FUNCTION_BLOCK SKILL_Gate (* Command authority for one skill: procedure calls only while the unit runs; OPC UA commands only from the occupation owner outside Production; unit control always *)
  (* Standard: 61499-2 *)
  (* Version 2.0, 2026-09-27, Project contributors, Filling cell reference model *)
  PACKAGE fillingcell;
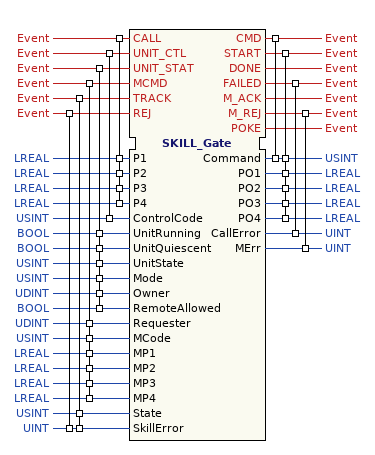
  EVENT_INPUT
    CALL WITH P1, P2, P3, P4;
    UNIT_CTL WITH ControlCode;
    UNIT_STAT WITH UnitRunning, UnitQuiescent, UnitState, Mode, Owner, RemoteAllowed;
    MCMD WITH Requester, MCode, MP1, MP2, MP3, MP4;
    TRACK WITH State, SkillError;
    REJ WITH SkillError;
  END_EVENT
  EVENT_OUTPUT
    CMD WITH Command;
    START WITH Command, PO1, PO2, PO3, PO4;
    DONE;
    FAILED WITH CallError;
    M_ACK;
    M_REJ WITH MErr;
    POKE;
  END_EVENT
  VAR_INPUT
    P1 : LREAL;
    P2 : LREAL;
    P3 : LREAL;
    P4 : LREAL;
    ControlCode : USINT;
    UnitRunning : BOOL;
    UnitQuiescent : BOOL;
    UnitState : USINT;
    Mode : USINT;
    Owner : UDINT;
    RemoteAllowed : BOOL;
    Requester : UDINT;
    MCode : USINT;
    MP1 : LREAL;
    MP2 : LREAL;
    MP3 : LREAL;
    MP4 : LREAL;
    State : USINT := 4;
    SkillError : UINT;
  END_VAR
  VAR_OUTPUT
    Command : USINT;
    PO1 : LREAL;
    PO2 : LREAL;
    PO3 : LREAL;
    PO4 : LREAL;
    CallError : UINT;
    MErr : UINT;
  END_VAR
  VAR
    CallPending : BOOL;
    PendingStart : BOOL;
    MPending : BOOL;
    ManualOK : BOOL;
    Valid : BOOL;
  END_VAR
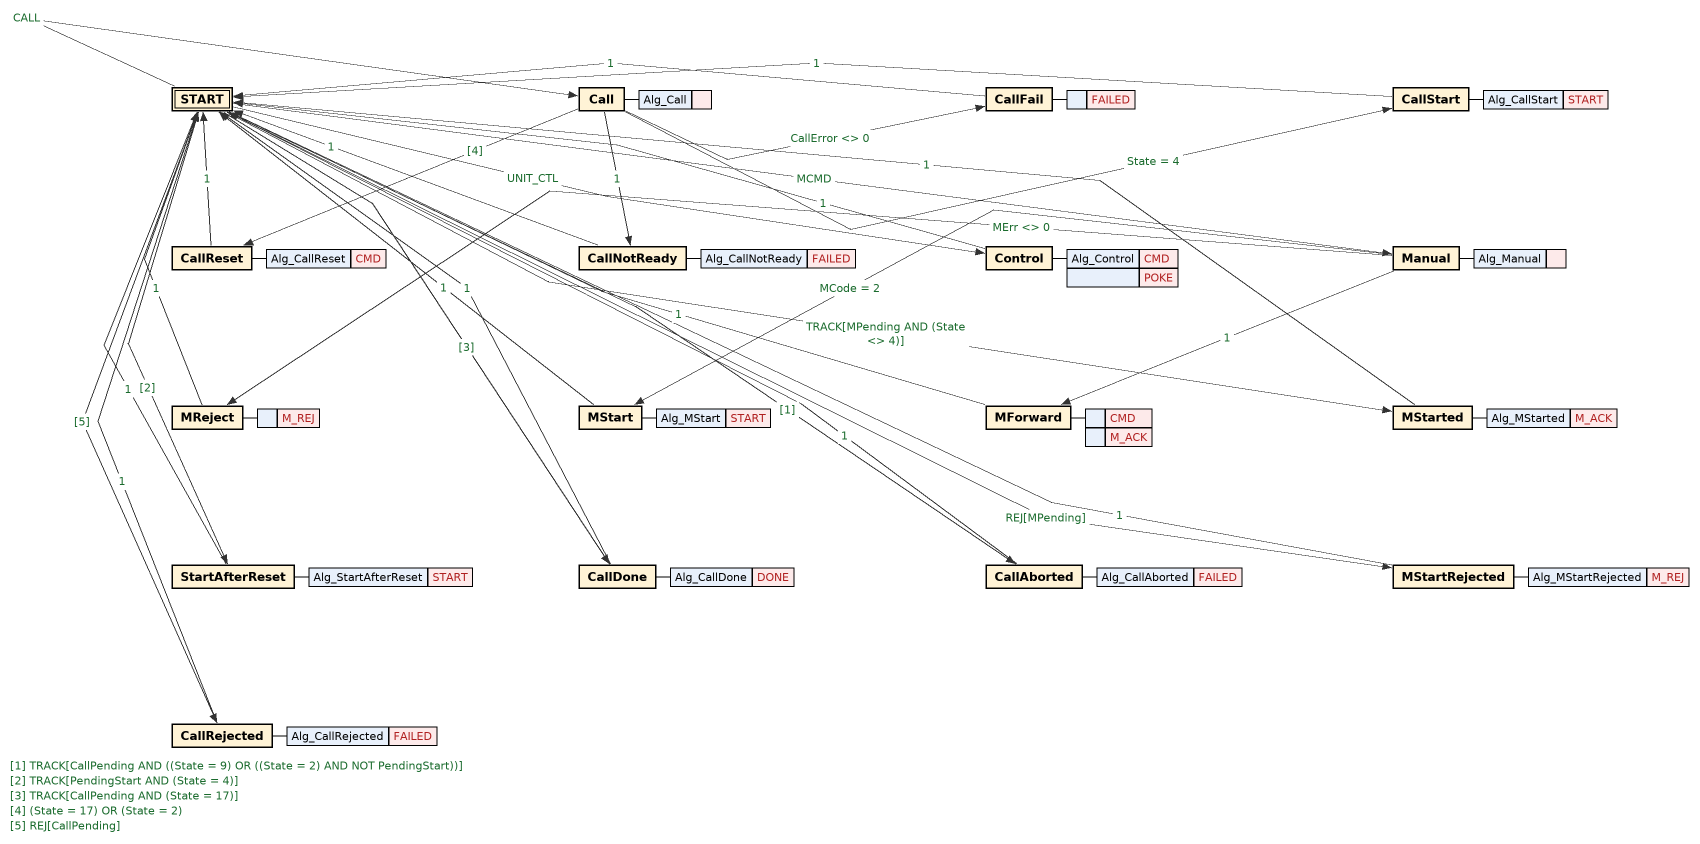
  EC_STATES
    START;
    Call : Alg_Call;
    CallFail : -> FAILED;
    CallStart : Alg_CallStart -> START;
    CallReset : Alg_CallReset -> CMD;
    CallNotReady : Alg_CallNotReady -> FAILED;
    Control : Alg_Control -> CMD, -> POKE;
    Manual : Alg_Manual;
    MReject : -> M_REJ;
    MStart : Alg_MStart -> START;
    MForward : -> CMD, -> M_ACK;
    MStarted : Alg_MStarted -> M_ACK;
    StartAfterReset : Alg_StartAfterReset -> START;
    CallDone : Alg_CallDone -> DONE;
    CallAborted : Alg_CallAborted -> FAILED;
    MStartRejected : Alg_MStartRejected -> M_REJ;
    CallRejected : Alg_CallRejected -> FAILED;
  END_STATES
  EC_TRANSITIONS
    START TO Call := CALL;
    Call TO CallFail := CallError <> 0;
    Call TO CallStart := State = 4;
    Call TO CallReset := (State = 17) OR (State = 2);
    Call TO CallNotReady := 1;
    CallFail TO START := 1;
    CallStart TO START := 1;
    CallReset TO START := 1;
    CallNotReady TO START := 1;
    START TO Control := UNIT_CTL;
    Control TO START := 1;
    START TO Manual := MCMD;
    Manual TO MReject := MErr <> 0;
    Manual TO MStart := MCode = 2;
    Manual TO MForward := 1;
    MReject TO START := 1;
    MStart TO START := 1;
    MForward TO START := 1;
    START TO MStarted := TRACK[MPending AND (State <> 4)];
    START TO StartAfterReset := TRACK[PendingStart AND (State = 4)];
    START TO CallDone := TRACK[CallPending AND (State = 17)];
    START TO CallAborted := TRACK[CallPending AND ((State = 9) OR ((State = 2) AND NOT PendingStart))];
    START TO MStartRejected := REJ[MPending];
    START TO CallRejected := REJ[CallPending];
    MStarted TO START := 1;
    StartAfterReset TO START := 1;
    CallDone TO START := 1;
    CallAborted TO START := 1;
    MStartRejected TO START := 1;
    CallRejected TO START := 1;
  END_TRANSITIONS
  ALGORITHM Alg_Call IN ST:
CallError := 0;
IF NOT UnitRunning THEN CallError := 5;
ELSIF CallPending OR MPending THEN CallError := 6;
END_IF;
PO1 := P1;
PO2 := P2;
PO3 := P3;
PO4 := P4;
  END_ALGORITHM
  ALGORITHM Alg_CallStart IN ST:
CallPending := TRUE;
Command := 2;
  END_ALGORITHM
  ALGORITHM Alg_CallReset IN ST:
CallPending := TRUE;
PendingStart := TRUE;
Command := 1;
  END_ALGORITHM
  ALGORITHM Alg_CallNotReady IN ST:
CallError := 4;
  END_ALGORITHM
  ALGORITHM Alg_Control IN ST:
Command := ControlCode;
IF (ControlCode = 5) OR (ControlCode = 6) THEN PendingStart := FALSE; END_IF;
  END_ALGORITHM
  ALGORITHM Alg_Manual IN ST:
MErr := 0;
Valid := FALSE;
CASE MCode OF
1: Valid := (State = 4) OR (State = 17) OR (State = 2);
2: Valid := State = 4;
3: Valid := State = 6;
4: Valid := State = 11;
5: Valid := (State = 4) OR (State = 6) OR (State = 11) OR (State = 17);
6: Valid := (State = 4) OR (State = 6) OR (State = 11) OR (State = 17) OR (State = 2);
7: Valid := State = 9;
END_CASE;
ManualOK := RemoteAllowed AND (Requester = Owner) AND (Requester <> 0) AND (Mode <> 0) AND NOT CallPending AND NOT MPending;
IF MCode = 2 THEN ManualOK := ManualOK AND UnitQuiescent AND (UnitState <> 9); END_IF;
IF NOT ManualOK THEN MErr := 5;
ELSIF NOT Valid THEN MErr := 4;
END_IF;
Command := MCode;
PO1 := MP1;
PO2 := MP2;
PO3 := MP3;
PO4 := MP4;
  END_ALGORITHM
  ALGORITHM Alg_MStart IN ST:
MPending := TRUE;
  END_ALGORITHM
  ALGORITHM Alg_MStarted IN ST:
MPending := FALSE;
  END_ALGORITHM
  ALGORITHM Alg_StartAfterReset IN ST:
PendingStart := FALSE;
Command := 2;
  END_ALGORITHM
  ALGORITHM Alg_CallDone IN ST:
CallPending := FALSE;
  END_ALGORITHM
  ALGORITHM Alg_CallAborted IN ST:
CallPending := FALSE;
PendingStart := FALSE;
CallError := SkillError;
IF CallError = 0 THEN CallError := 7; END_IF;
  END_ALGORITHM
  ALGORITHM Alg_MStartRejected IN ST:
MPending := FALSE;
MErr := SkillError;
  END_ALGORITHM
  ALGORITHM Alg_CallRejected IN ST:
CallPending := FALSE;
CallError := SkillError;
  END_ALGORITHM
END_FUNCTION_BLOCK
